(* CODESYS project CmpEmiconLog.library
   Author: Emicon
   Title: EmiconLog
   Version: 3.5.17.21
   Placeholder: PlaceholderTemplate
   DocFormat: reStructuredText
   Description: Emicon logging functionality
   Company: Emicon
   LanguageModelAttribute: qualified-access-only
   DefaultNamespace: EmLog

Project tree, tasks and I/O mapping:
  function write_sys_log [ST]
  function write_ts_log [ST]
  function write_ti_log [ST]
  function clr_sys_log [ST]
  function create_log_files [ST]
  function get_next_log_item [ST]
*)

// write_sys_log
FUNCTION write_sys_log : UDINT
VAR_INPUT
	bySeverity	: BYTE;  // Уровень важности. ОДЗ: 0..7
	byClassId 	: BYTE;	 // Класс (модуль, блок и т.п.), инициировавший запись в системный журнал. ОДЗ: 0...255
	byEvent		: BYTE;  // Cобытие. ОДЗ: 0...31
	dwArgs 		: DWORD; // Аргументы. Массив из 4х байт.
END_VAR
VAR
END_VAR

END_FUNCTION

// write_ts_log
{attribute 'hide'}
FUNCTION write_ts_log : UDINT
VAR_INPUT
	byClassId: BYTE;
	pbyData : POINTER TO BYTE;
END_VAR
VAR
END_VAR

END_FUNCTION

// write_ti_log
{attribute 'hide'}
FUNCTION write_ti_log : UDINT
VAR_INPUT
	byClassId: BYTE;
	pbyData : POINTER TO BYTE;
END_VAR
VAR
END_VAR

END_FUNCTION

// clr_sys_log
FUNCTION clr_sys_log : UDINT
VAR_INPUT
END_VAR
VAR
END_VAR

END_FUNCTION

// create_log_files
FUNCTION create_log_files : DINT
VAR_INPUT
END_VAR
VAR
END_VAR

END_FUNCTION

// get_next_log_item
{attribute 'hide'}
FUNCTION get_next_log_item : int
VAR_INPUT
	get_first : BOOL;
	log_str : POINTER TO STRING;
END_VAR
VAR
END_VAR

END_FUNCTION
